{attribute 'qualified_only'}
{attribute 'strict'}
{attribute 'to_string'}
TYPE E_MachinePreparationErrorCode :
(
    None                    := 16#0000,
    AxisNotConfigured       := 16#C101,
    AxisReadyTimeout        := 16#C102,
    StandbyMotionTimeout    := 16#C103,
    GripperOpenFailed       := 16#C104,
    InvalidProcessStep      := 16#C1FF,
    AxisAlarmBase           := 16#C200,
    AxisCommandFailureBase  := 16#C300
) UDINT;
END_TYPE

(* stored: Version 1.1.0.1, ProductVersion 3.1.4026.20
   DUT E_MachinePreparationErrorCode: Id {781694b1-3bc0-4d13-b399-54c17f011145} *)
